// SIMATIC STEP 7 (V5.x) project TankAndMixer
// CPU: CPU 315-2 DP
// station: Hardware
// station: SIMATIC 300(1)
// station: P_ADR_BUS
// program: S7 Program(1)

SYMBOL_TABLE
"START_BUTTON"	I 0.0	BOOL
"STOP"	I 0.1	BOOL
"STARTBIT"	M 0.0	BOOL
"STOPBIT"	M 0.1	BOOL
"MIXEROFFTRIGGER"	M 0.2	BOOL
"PUMP1"	Q 0.0	BOOL
"PUMP2"	Q 0.1	BOOL
"MIXER"	Q 0.2	BOOL
"PUMP3"	Q 0.3	BOOL
"P1TIMER"	T 0	TIMER
"MIXERTIMER"	T 1	TIMER
"P2TIMER"	T 2	TIMER
"P3TIMER"	T 3	TIMER
END_SYMBOL_TABLE

ORGANIZATION_BLOCK OB 1
TITLE = "Main Program Sweep (Cycle)"
VERSION : 0.1
VAR_TEMP
  OB1_EV_CLASS : BYTE ;	//Bits 0-3 = 1 (Coming event), Bits 4-7 = 1 (Event class 1)
  OB1_SCAN_1 : BYTE ;	//1 (Cold restart scan 1 of OB 1), 3 (Scan 2-n of OB 1)
  OB1_PRIORITY : BYTE ;	//Priority of OB Execution
  OB1_OB_NUMBR : BYTE ;	//1 (Organization block 1, OB1)
  OB1_RESERVED_1 : BYTE ;	//Reserved for system
  OB1_RESERVED_2 : BYTE ;	//Reserved for system
  OB1_PREV_CYCLE : INT ;	//Cycle time of previous OB1 scan (milliseconds)
  OB1_MIN_CYCLE : INT ;	//Minimum cycle time of OB1 (milliseconds)
  OB1_MAX_CYCLE : INT ;	//Maximum cycle time of OB1 (milliseconds)
  OB1_DATE_TIME : DATE_AND_TIME ;	//Date and time OB1 started
END_VAR
BEGIN
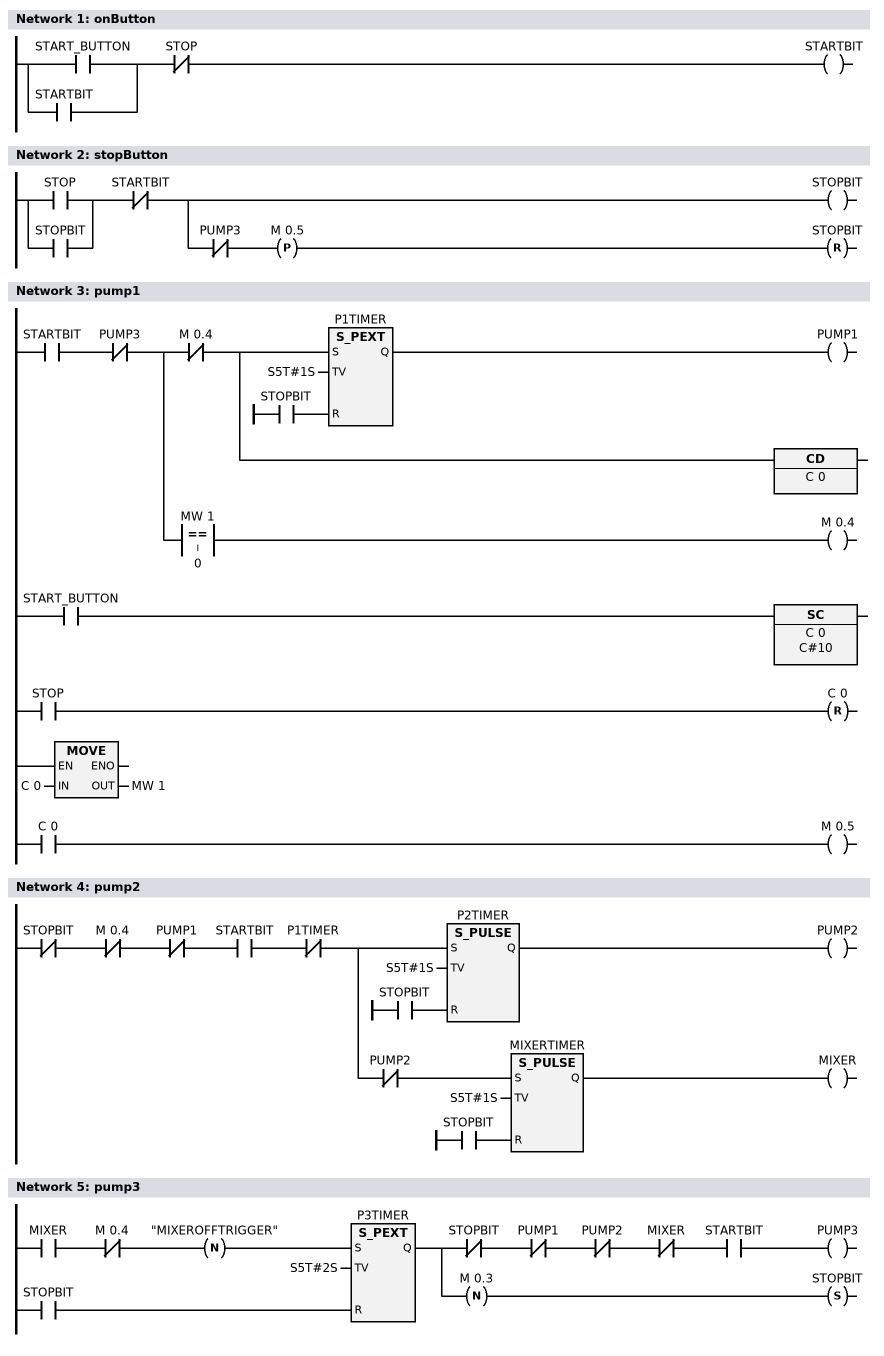
NETWORK
TITLE = onButton
      A(;
      O     "START_BUTTON";
      O     "STARTBIT";
      );
      AN    "STOP";
      =     "STARTBIT";
NETWORK
TITLE = stopButton
      A(;
      O     "STOP";
      O     "STOPBIT";
      );
      AN    "STARTBIT";
      =     L 20.0;
      A     L 20.0;
      BLD   102;
      =     "STOPBIT";
      A     L 20.0;
      AN    "PUMP3";
      FP    M 0.5;
      R     "STOPBIT";
NETWORK
TITLE = pump1
      A     "STARTBIT";
      AN    "PUMP3";
      =     L 20.0;
      A     L 20.0;
      AN    M 0.4;
      =     L 20.1;
      A     L 20.1;
      L     S5T#1S;
      SE    "P1TIMER";
      A     "STOPBIT";
      R     "P1TIMER";
      NOP   0;
      NOP   0;
      A     "P1TIMER";
      =     "PUMP1";
      A     L 20.1;
      CD    C 0;
      BLD   101;
      A     "START_BUTTON";
      L     C#10;
      S     C 0;
      A     "STOP";
      R     C 0;
      L     C 0;
      T     MW 1;
      NOP   0;
      A     C 0;
      =     M 0.5;
      A     L 20.0;
      A(;
      L     MW 1;
      L     0;
      ==I;
      );
      =     M 0.4;
NETWORK
TITLE = pump2
      AN    "STOPBIT";
      AN    M 0.4;
      AN    "PUMP1";
      A     "STARTBIT";
      AN    "P1TIMER";
      =     L 20.0;
      A     L 20.0;
      L     S5T#1S;
      SP    "P2TIMER";
      A     "STOPBIT";
      R     "P2TIMER";
      NOP   0;
      NOP   0;
      A     "P2TIMER";
      =     "PUMP2";
      A     L 20.0;
      AN    "PUMP2";
      L     S5T#1S;
      SP    "MIXERTIMER";
      A     "STOPBIT";
      R     "MIXERTIMER";
      NOP   0;
      NOP   0;
      A     "MIXERTIMER";
      =     "MIXER";
NETWORK
TITLE = pump3
      A     "MIXER";
      AN    M 0.4;
      FN    "MIXEROFFTRIGGER";
      L     S5T#2S;
      SE    "P3TIMER";
      A     "STOPBIT";
      R     "P3TIMER";
      NOP   0;
      NOP   0;
      A     "P3TIMER";
      =     L 20.0;
      A     L 20.0;
      AN    "STOPBIT";
      AN    "PUMP1";
      AN    "PUMP2";
      AN    "MIXER";
      A     "STARTBIT";
      =     "PUMP3";
      A     L 20.0;
      FN    M 0.3;
      S     "STOPBIT";
END_ORGANIZATION_BLOCK
